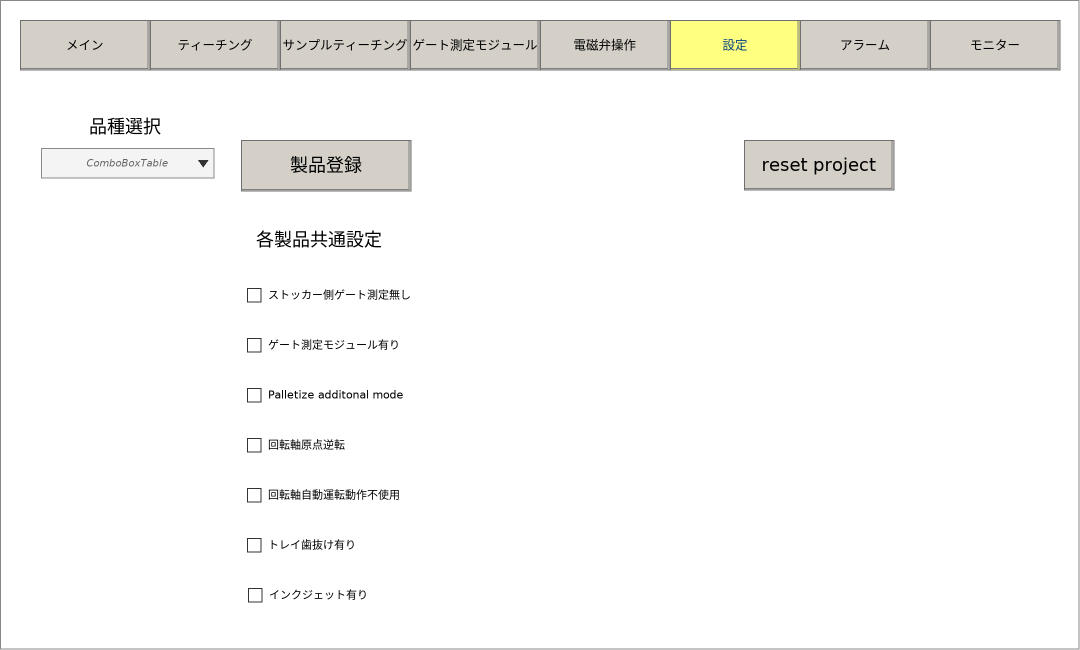
VISUALIZATION s_setting  // 1080x650
    Rectangle (0,0 1080x650)
    Label (50,112 150x30), "品種選択"
    ComboBoxTable (41,148 173x30), variable: gvl_param.var_currentProductID, data array: gvl_visu.var_in_currentProduct
        p3854506369: gvl_visu.var_in_currentProduct[INDEX]
    Checkbox (245,280 400x30), "ストッカー側ゲート測定無し", variable: gvl_visu.flg_btn_gateMeasurementIsNone
    Checkbox (245,330 400x30), "ゲート測定モジュール有り", variable: gvl_visu.flg_btn_usingMeasurementSystem
    Button (241,140 170x51), "製品登録"
        OnMouseClick: change screen: s_addNewProduct
    Checkbox (245,380 400x30), "Palletize additonal mode", variable: gvl_visu.var_dev_palletizingMode
    Button (20,20 130x50), "メイン"
        OnMouseClick: change screen: s_auto
    Button (150,20 130x50), "ティーチング"
        OnMouseClick: change screen: s_teaching1
    Button (670,20 130x50), "設定"
        OnMouseClick: change screen: s_setting
    Button (540,20 130x50), "電磁弁操作"
        OnMouseClick: change screen: s_manual
    Button (410,20 130x50), "ゲート測定モジュール"
        OnMouseClick: change screen: s_gm_teaching
    Button (800,20 130x50), "アラーム", colour toggle: gvl_io.flg_signalTowerRed
        OnMouseClick: change screen: s_alarm
    Button (280,20 130x50), "サンプルティーチング"
        OnMouseClick: change screen: s_sample
    Button (744,140 150x50), "reset project"
        OnMouseClick: OpenDialog Dialog=d_resetProject, OpenModal=True, OpenCentered=True
    Checkbox (245,430 400x30), "回転軸原点逆転", variable: gvl_visu.flg_btn_rotaryReversal
    Checkbox (245,480 400x30), "回転軸自動運転動作不使用", variable: gvl_visu.flg_btn_RotaryIsNotUse
    Checkbox (245,530 400x30), "トレイ歯抜け有り", variable: gvl_visu.flg_missingParts
    Checkbox (246,580 400x30), "インクジェット有り", variable: gvl_visu.flg_usingTimeStamp
    Button (930,20 130x50), "モニター"
        OnMouseClick: change screen: s_monitor
    Label (253,213 189x54), "各製品共通設定"
END_VISUALIZATION

(* stored: Version 1.1.0.1, ProductVersion 3.1.4024.11
   Visu s_setting: Id {909b483f-3287-4372-a805-cd82e146060b} *)
